// SIMATIC S7-200 project (STEP 7-Micro/WIN), CPU 224XP REL 02.01

SYMBOL_TABLE USUARIO1
PARO             I0.0
MARCHA           I0.1
LAMPARA          Q0.0
END_SYMBOL_TABLE

ORGANIZATION_BLOCK PRINCIPAL:OB1
TITLE=COMENTARIOS DEL PROGRAMA
BEGIN
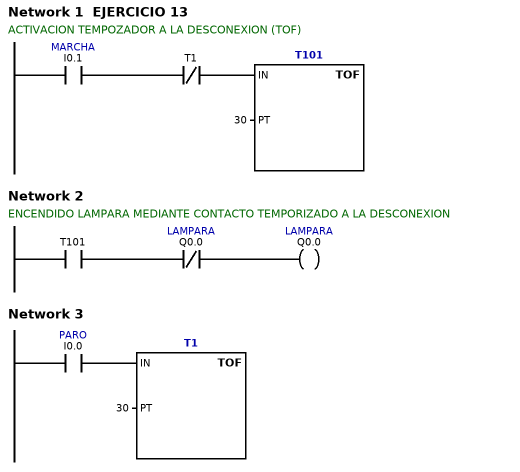
Network 1 // EJERCICIO 13
// ACTIVACION TEMPOZADOR A LA DESCONEXION (TOF)
// (network saved uncompiled; LAD cells follow)
// row 0: c0 -| |- MARCHA:I0.1  c1 -|/|- T1  c2 [TOF T101 IN:=power@row0, PT:=30]
// row 1: c2 [box]
Network 2
// ENCENDIDO LAMPARA MEDIANTE CONTACTO TEMPORIZADO A LA DESCONEXION  
// (network saved uncompiled; LAD cells follow)
// row 0: c0 -| |- T101  c1 -|/|- LAMPARA:Q0.0  c2 -( ) LAMPARA:Q0.0
Network 3
// (network saved uncompiled; LAD cells follow)
// row 0: c0 -| |- PARO:I0.0  c1 [TOF T1 IN:=power@row0, PT:=30]
// row 1: c1 [box]
END_ORGANIZATION_BLOCK
